{attribute 'GeneratedUsingTerminal: EPP1111-0000-0016'}
{attribute addProperty BoxType "EPP1111-0000-0016"}
{attribute addProperty Id "IDAT %I*UINT2"}
{attribute addProperty CRC "130667151"}
{attribute addProperty Size "2"}
TYPE ID_Inputs_07C9D28F EXTENDS InputBase_8311D824 :
STRUCT
	{attribute addProperty Name "ID"}
	ID AT %I* : UINT;
END_STRUCT
END_TYPE

(* stored: Version 1.2.0.0, ProductVersion 3.1.4024.9
   DUT ID_Inputs_07C9D28F: Id {01fac5d3-a819-4070-bfa0-099ae88ae87d} *)
